(* IEC 61131-3 sources: CodesysTest/alpha/export/PackML/Pregis/StateMachine, 18 files *)

(* ---- Aborted.pou.st ---- *)
(*#-#-#-#-#-#-#-#-#-#---Declaration---#-#-#-#-#-#-#-#-#-#-#-#-#*)

FUNCTION_BLOCK Aborted EXTENDS BaseState
VAR_INPUT
END_VAR
VAR_OUTPUT
END_VAR
VAR
END_VAR

(* ---- Aborting.pou.st ---- *)
(*#-#-#-#-#-#-#-#-#-#---Declaration---#-#-#-#-#-#-#-#-#-#-#-#-#*)

FUNCTION_BLOCK Aborting EXTENDS BaseState
VAR_INPUT
END_VAR
VAR_OUTPUT
END_VAR
VAR
END_VAR

(* ---- BaseState.pou.st ---- *)
(*#-#-#-#-#-#-#-#-#-#---Declaration---#-#-#-#-#-#-#-#-#-#-#-#-#*)

FUNCTION_BLOCK BaseState
VAR_INPUT
	Begin : BOOL := FALSE;
END_VAR
VAR_OUTPUT
	End : BOOL := False;
END_VAR
VAR
END_VAR

(* ---- Clearing.pou.st ---- *)
(*#-#-#-#-#-#-#-#-#-#---Declaration---#-#-#-#-#-#-#-#-#-#-#-#-#*)

FUNCTION_BLOCK Clearing EXTENDS BaseState
VAR_INPUT
END_VAR
VAR_OUTPUT
END_VAR
VAR
END_VAR

(* ---- Complete.pou.st ---- *)
(*#-#-#-#-#-#-#-#-#-#---Declaration---#-#-#-#-#-#-#-#-#-#-#-#-#*)

FUNCTION_BLOCK Complete EXTENDS BaseState
VAR_INPUT
END_VAR
VAR_OUTPUT
END_VAR
VAR
END_VAR

(* ---- Completing.pou.st ---- *)
(*#-#-#-#-#-#-#-#-#-#---Declaration---#-#-#-#-#-#-#-#-#-#-#-#-#*)

FUNCTION_BLOCK Completing EXTENDS BaseState
VAR_INPUT
END_VAR
VAR_OUTPUT
END_VAR
VAR
END_VAR

(* ---- Execute.pou.st ---- *)
(*#-#-#-#-#-#-#-#-#-#---Declaration---#-#-#-#-#-#-#-#-#-#-#-#-#*)

FUNCTION_BLOCK Execute EXTENDS BaseState
VAR_INPUT
END_VAR
VAR_OUTPUT
END_VAR
VAR
END_VAR

(* ---- Held.pou.st ---- *)
(*#-#-#-#-#-#-#-#-#-#---Declaration---#-#-#-#-#-#-#-#-#-#-#-#-#*)

FUNCTION_BLOCK Held
VAR_INPUT
END_VAR
VAR_OUTPUT
END_VAR
VAR
END_VAR

(* ---- Holding.pou.st ---- *)
(*#-#-#-#-#-#-#-#-#-#---Declaration---#-#-#-#-#-#-#-#-#-#-#-#-#*)

FUNCTION_BLOCK Holding EXTENDS BaseState
VAR_INPUT
END_VAR
VAR_OUTPUT
END_VAR
VAR
END_VAR

(* ---- Idle.pou.st ---- *)
(*#-#-#-#-#-#-#-#-#-#---Declaration---#-#-#-#-#-#-#-#-#-#-#-#-#*)

FUNCTION_BLOCK Idle EXTENDS BaseState
VAR_INPUT
END_VAR
VAR_OUTPUT
END_VAR
VAR
END_VAR

(* ---- Resetting.pou.st ---- *)
(*#-#-#-#-#-#-#-#-#-#---Declaration---#-#-#-#-#-#-#-#-#-#-#-#-#*)

FUNCTION_BLOCK Resetting EXTENDS BaseState
VAR_INPUT
END_VAR
VAR_OUTPUT
END_VAR
VAR
END_VAR

(* ---- Starting.pou.st ---- *)
(*#-#-#-#-#-#-#-#-#-#---Declaration---#-#-#-#-#-#-#-#-#-#-#-#-#*)

FUNCTION_BLOCK Starting EXTENDS BaseState
VAR_INPUT
END_VAR
VAR_OUTPUT
END_VAR
VAR
END_VAR

(* ---- Stopped.pou.st ---- *)
(*#-#-#-#-#-#-#-#-#-#---Declaration---#-#-#-#-#-#-#-#-#-#-#-#-#*)

FUNCTION_BLOCK Stopped EXTENDS BaseState
VAR_INPUT
END_VAR
VAR_OUTPUT
END_VAR
VAR
END_VAR

(* ---- Stopping.pou.st ---- *)
(*#-#-#-#-#-#-#-#-#-#---Declaration---#-#-#-#-#-#-#-#-#-#-#-#-#*)

FUNCTION_BLOCK Stopping EXTENDS BaseState
VAR_INPUT
END_VAR
VAR_OUTPUT
END_VAR
VAR
END_VAR

(* ---- Suspended.pou.st ---- *)
(*#-#-#-#-#-#-#-#-#-#---Declaration---#-#-#-#-#-#-#-#-#-#-#-#-#*)

FUNCTION_BLOCK Suspended EXTENDS BaseState
VAR_INPUT
END_VAR
VAR_OUTPUT
END_VAR
VAR
END_VAR

(* ---- Suspending.pou.st ---- *)
(*#-#-#-#-#-#-#-#-#-#---Declaration---#-#-#-#-#-#-#-#-#-#-#-#-#*)

FUNCTION_BLOCK Suspending EXTENDS BaseState
VAR_INPUT
END_VAR
VAR_OUTPUT
END_VAR
VAR
END_VAR

(* ---- Unholding.pou.st ---- *)
(*#-#-#-#-#-#-#-#-#-#---Declaration---#-#-#-#-#-#-#-#-#-#-#-#-#*)

FUNCTION_BLOCK Unholding EXTENDS BaseState
VAR_INPUT
END_VAR
VAR_OUTPUT
END_VAR
VAR
END_VAR

(* ---- Unsuspending.pou.st ---- *)
(*#-#-#-#-#-#-#-#-#-#---Declaration---#-#-#-#-#-#-#-#-#-#-#-#-#*)

FUNCTION_BLOCK Unsuspending EXTENDS BaseState
VAR_INPUT
END_VAR
VAR_OUTPUT
END_VAR
VAR
END_VAR
